INTERFACE PUBLIC HoldingCommands EXTENDS RunningStateCommands, ActionStateCommands

END_INTERFACE

(* stored: Version 1.1.0.1, ProductVersion 3.1.4026.18
   Itf HoldingCommands: Id {af08fee2-ed8e-0073-1bb5-3408d155c093} *)
